FUNCTION_BLOCK RampDown
VAR_INPUT
	IN: BOOL;
	RampDownTime: TIME;
	Ramp_lowerLimit: REAL;
	Ramp_upperLimit: REAL;
	PLC_CYCLE_TIME_ms: REAL;
END_VAR
VAR_IN_OUT
	output: REAL;
END_VAR
VAR_OUTPUT
	InProgress: BOOL;	
END_VAR
VAR
	rampDown: REAL;
	x: REAL;
	init: BOOL;
END_VAR


	IF IN AND (RampDownTime > T#0S) AND (PLC_CYCLE_TIME_ms > 0) THEN
		IF NOT init THEN
			init	:=	TRUE;
			InProgress	:=	TRUE;
			rampDown	:=	TIME_TO_REAL(RampDownTime);		
			x		:=	PLC_CYCLE_TIME_ms / rampDown;
			x		:=	(Ramp_upperLimit - Ramp_lowerLimit) * x;
		END_IF
		
		IF (output > Ramp_lowerLimit) AND (InProgress) THEN
			output		:=	output - x;
		ELSE
			output		:=	Ramp_lowerLimit;
			InProgress	:=	FALSE;
		END_IF
		
	ELSE
		InProgress 	:=	FALSE;	
		init		:=	FALSE;
	END_IF

END_FUNCTION_BLOCK

(* stored: Version 1.1.0.1, ProductVersion 3.1.4024.13
   POU RampDown: Id {0cc193c6-3e00-4562-a9a9-f327daf82b5e}, SpecialFunc None *)
